(*

.. <legal notes>

legal notes
=================
| SPDX-FileCopyrightText: © 2026 Oleksandr Tiutyk <trofimich@gmail.com>
| SPDX-License-Identifier: LGPL-3.0-only
| For details check: LGPL-3.0-only_

.. _LGPL-3.0-only: https://www.gnu.org/licenses/lgpl-3.0.en.html

.. </legal notes>

*)

PROGRAM UsignedInt16Helper
VAR CONSTANT
	MIN_VALUE : UINT := 0;
	MAX_VALUE : UINT := 65_535;
END_VAR
VAR
	_ClassName : STRING := __POUNAME();
END_VAR

{attribute 'monitoring' := 'call'}
PROPERTY ClassName : STRING
GET
ClassName := _ClassName;
END_GET
END_PROPERTY

{attribute 'monitoring' := 'call'}
PROPERTY NamespaceName : STRING
GET
NamespaceName := CurrentNamespace.Name;
END_GET
END_PROPERTY

END_PROGRAM

(* stored: Version 1.1.0.1
   POU UsignedInt16Helper: Id {359c1cce-ae3b-4104-951e-6498f593d0f2}, SpecialFunc None
   Property ClassName: Id {e28f3e6b-f8ef-4f8f-aaca-b868322c98eb}
   Get Get: Id {91af5dcb-ef23-4bee-8853-6d037edab072}
   Property NamespaceName: Id {de673b86-8af7-471b-8059-506452281cca}
   Get Get: Id {c5c97b87-3837-4e30-b5d4-b8fd59f60799} *)
